///#########################################################
///Function block to write parameter in Nc.
///
/// Library:
/// Tc2_MC2.lib
/// Tc2_System.lib
///
/// Global Variables:
///
/// Data types:
///
/// External functions:
///
/// History:
/// 2014-02-05  v1.00   NB  Release code.
///
/// Known bugs:
///
///
///
///###########################################################
FUNCTION_BLOCK FB_WriteFloatParameter
VAR_INPUT
    bExecute: BOOL;
    ///16#4000=Axisdata, 16#5000=Encoderdata, 16#6000=Controldata, 16#7000=Drivedata
    nDeviceGroup: UDINT;
    nIndexOffset: UDINT;
    nData: LREAL;
END_VAR
VAR_OUTPUT
    bBusy: BOOL;
    bDone: BOOL;
    bError: BOOL;
    nErrorId: UDINT;
END_VAR
VAR_IN_OUT
    Axis: AXIS_REF;
END_VAR
VAR
    nState: UINT;
    fbADSWRITE: ADSWRITE;
END_VAR

(*Sequence to write parameter in Nc*)
CASE nState OF
0:  (*Start sequence. Wait until bExecute is TRUE*)
    IF bExecute THEN
        bBusy:=TRUE;
        bError:=FALSE;
        nErrorId:=0;
        nState:=10;
    END_IF

10: (*Write parameter in Nc*)
    fbADSWRITE(
        PORT:=500,
        IDXGRP:=nDeviceGroup+Axis.NcToPlc.AxisId,
        IDXOFFS:=nIndexOffset,
        LEN:=SIZEOF(nData),
        SRCADDR:=ADR(nData),
        WRITE:=TRUE);

    (*Wait until it's done or if an error occurs*)
    IF NOT fbADSWRITE.ERR THEN
        IF NOT fbADSWRITE.BUSY THEN
            fbADSWRITE(WRITE:=FALSE);
            nState:=20;
        END_IF
    ELSE
        nErrorId:=fbADSWRITE.ERRID;
        nState:=999;
    END_IF

20: (*Sequense is done. Waits until bExecute is FALSE*)
    bBusy:=FALSE;
    bDone:=TRUE;
    IF NOT bExecute THEN
        bDone:=FALSE;
        nState:=0;
    END_IF

999: (*Error in sequence*)
    bError:=TRUE;
    bBusy:=FALSE;
    bDone:=FALSE;
    fbADSWRITE(WRITE:=FALSE);
    IF NOT bExecute THEN
        nState:=0;
    END_IF

END_CASE

END_FUNCTION_BLOCK

(* stored: Version 1.1.0.1, ProductVersion 3.1.4024.6
   POU FB_WriteFloatParameter: Id {8d98c0d3-e029-4bc1-bb0d-006a7c407e39}, SpecialFunc None *)
